//{attribute 'qualified_only'}
//{attribute 'strict'}
{attribute 'to_string'}

TYPE E_Util_Service_Sts :
(
	PowerUp		:= 0,
	Ready		:= 1,
	Running		:= 2,
	Faulted		:= 9
);
END_TYPE

(* stored: Version 1.1.0.1, ProductVersion 3.1.4024.12
   DUT E_Util_Service_Sts: Id {ed0539d3-9462-4157-8bfe-81ced6969cf9} *)
